RoboDK station: movimiento_mocap16ene.rdk

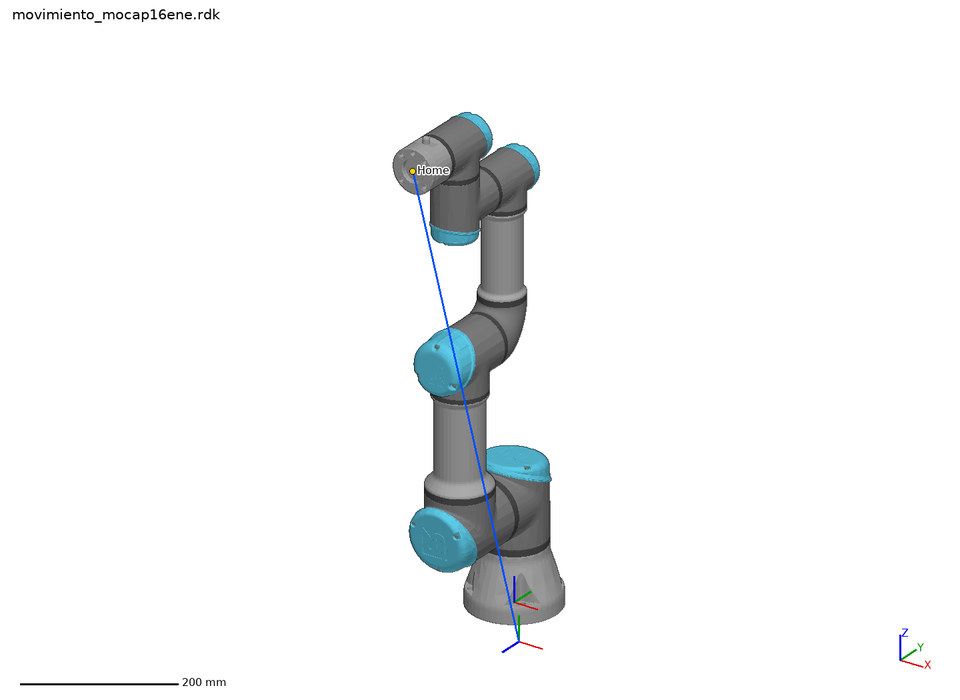
[picture v0: the station drawn from its stored meshes, robots at their saved joint values, targets as dots, program paths as lines]
Station movimiento_mocap (saved by RoboDK 5.5.2). Poses are relative to the parent item; angles as X-Y-Z fixed-axis rotations.
  - frame UR3e Base at (0, 0, 0) mm
    - robot UR3e: 6 axes, payload 3 kg, reach 500 mm, repeatability 0.03 mm, weight 11 kg
        modified DH rows (alpha deg, a mm, theta deg, d mm): 0, 0, 0, 151.9; 90, 0, 180, 0; 0, 243.55, 0, 0; 0, 213.2, 0, 131.05; -90, 0, 0, 85.35; 90, 0, 180, 92.1
        joint limits [-360, -360, -360, -360, -360, -360] to [360, 360, 360, 360, 360, 360]; home [0, -90, -90, 0, 90, 0]; saved at [0, -90, 0, -90, 0, 0]
    - frame B0 frame at (70, -90, 0) mm, rotated rx 90 ry 0 rz 0 deg
      - target Home (joint target) at (-70, 694, 133.15) mm, rotated rx 0 ry 0 rz 180 deg; joints [0, -90, 0, -90, 0, 0] of UR3e
      - target Target1 [record not read]
      - target Target2 [record not read]
      - target Home (joint target) at (-70, 694, 133.15) mm, rotated rx 0 ry 0 rz 180 deg; joints [0, -90, 0, -90, 0, 0] of UR3e
  - program My Prog (4 instructions, listed below)

--- program My Prog (robot UR3e) ---
  MoveJ (Home)
  MoveJ (Target1)
  MoveJ (Target2)
  MoveJ (Home)
